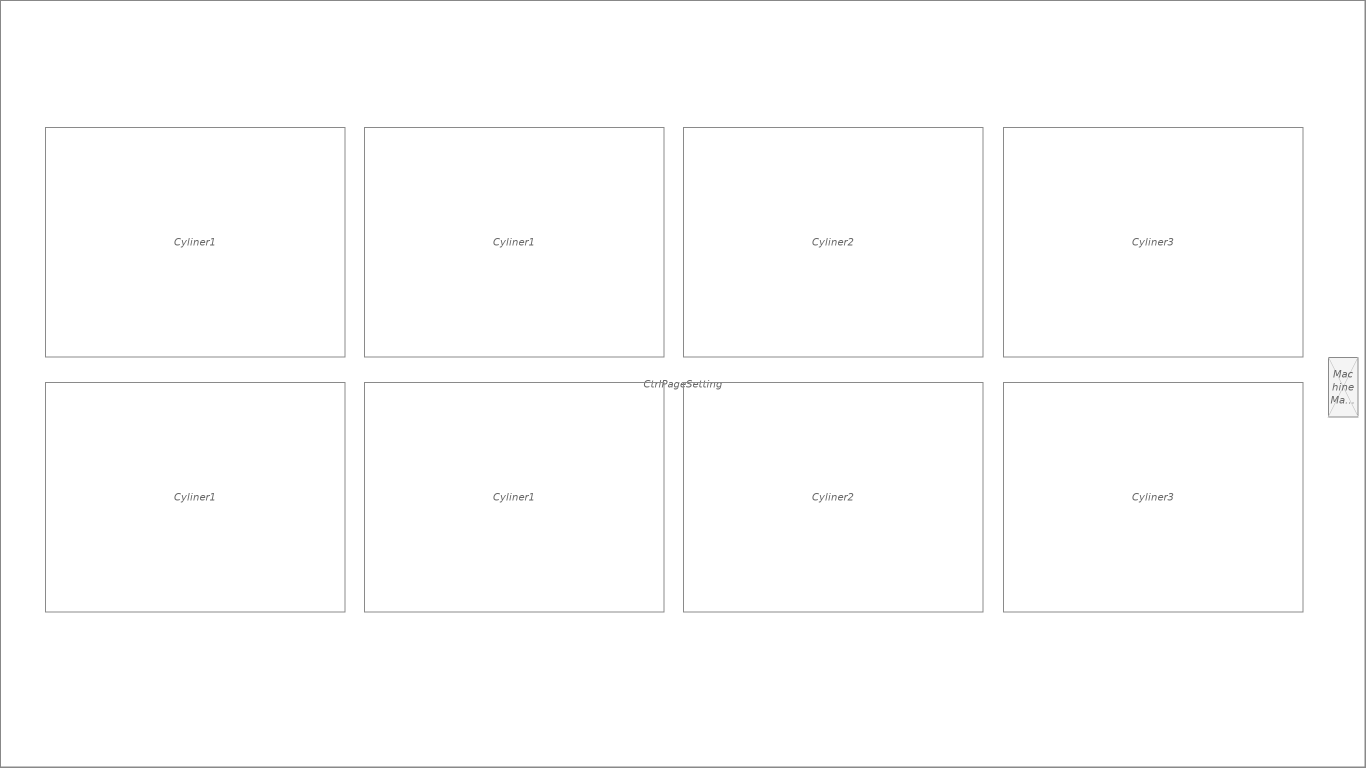
VISUALIZATION PageSetting_AcquireLoad  // 1366x768
    Frame (0,0 1366x768)
        shows CtrlPageSetting()
    Frame (45,127 300x230)
        shows Cyliner1(System := G_stSystem, Cylinder := G_arrCylinder[E_Cylinder.Line0Part], CylinderData := G_arrCylinderData[E_Cylinder.Line0Part])
    Frame (364,127 300x230)
        shows Cyliner1(System := G_stSystem, Cylinder := G_arrCylinder[E_Cylinder.Line0Prevent], CylinderData := G_arrCylinderData[E_Cylinder.Line0Prevent])
    Frame (45,382 300x230)
        shows Cyliner1(System := G_stSystem, Cylinder := G_arrCylinder[E_Cylinder.AcquirePrevent1], CylinderData := G_arrCylinderData[E_Cylinder.AcquirePrevent1])
    Frame (364,382 300x230)
        shows Cyliner1(System := G_stSystem, Cylinder := G_arrCylinder[E_Cylinder.AcquireLift], CylinderData := G_arrCylinderData[E_Cylinder.AcquireLift])
    Frame (683,382 300x230)
        shows Cyliner2(System := G_stSystem, Cylinder := G_arrCylinder[E_Cylinder.AcquirePush], CylinderData := G_arrCylinderData[E_Cylinder.AcquirePush])
    Frame (1003,382 300x230)
        shows Cyliner3(System := G_stSystem, Cylinder := G_arrCylinder[E_Cylinder.AcquireElevator], CylinderData := G_arrCylinderData[E_Cylinder.AcquireElevator])
    Frame (683,127 300x230)
        shows Cyliner2(System := G_stSystem, Cylinder := G_arrCylinder[E_Cylinder.Line0Push], CylinderData := G_arrCylinderData[E_Cylinder.Line0Push])
    Image (1328,357 30x60), image: MachineManage.ImagePool.next
        OnMouseClick: change screen: PageSetting_AcquireLoad_2
    Frame (1003,127 300x230)
        shows Cyliner3(System := G_stSystem, Cylinder := G_arrCylinder[E_Cylinder.Line0PushElevator], CylinderData := G_arrCylinderData[E_Cylinder.Line0PushElevator])
END_VISUALIZATION

(* stored: Version 1.1.0.1, ProductVersion 3.1.4024.3
   Visu PageSetting_AcquireLoad: Id {cab1f9ba-6338-4451-807c-87e43a0ff09a} *)
